{attribute 'qualified_only'}
{attribute 'strict'}
{attribute 'to_string'}
TYPE E_MIRROR_PROCESSOR_STEPS :
(
	INIT := 0,
	
	LOCATE_RIGHT_EDGE,
	
	LOCATE_TOP_EDGE,

	LOCATE_BOTTOM_EDGE,
	
	DRAW_POINTS,
	
	MAKE_DISPLAYABLE,
	
	DONE,
	
	ERROR,
	
	END
	
);
END_TYPE

(* stored: Version 1.1.0.1
   DUT E_MIRROR_PROCESSOR_STEPS: Id {b5e282f5-a97f-4c3e-8319-ed28edad8006} *)
